{attribute 'qualified_only'}
VAR_GLOBAL
	act: ARRAY[1..99] OF struct_SFC_Row;
END_VAR

(* stored: Version 1.1.0.1, ProductVersion 3.1.4024.12
   GVL S1sfc: Id {8efb6cdf-f37b-4370-be27-3ec30d1d8a87} *)
